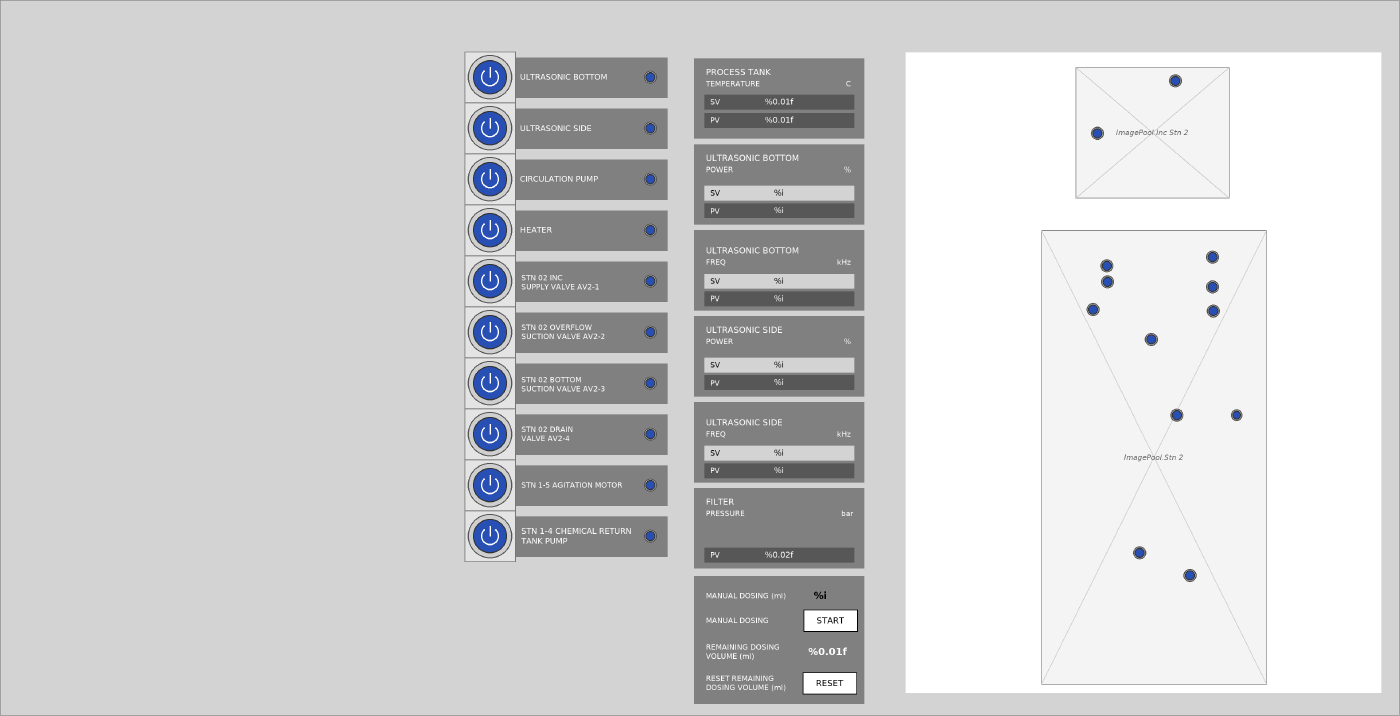
VISUALIZATION Manual_Station02  // 1920x983
    Rectangle (0,0 1920x983)
    Rectangle (1242,72 652x879)
    Image (1428,316 309x624), image: ImagePool.Stn 2
    RoundedRectangle (676,79 239x55)
    Label (710,98 163x16), "ULTRASONIC BOTTOM"
    Lamp1 (882,96 20x20), variable: ARdsMAP_HmiVariableStn[2].bProTankUsBtm_IND, style: Lamp-Lamp1-Blue
    PowerSwitch (637,71 70x70), variable: ARdsMAP_HmiVariableStn[2].bProTankUsBtm_PB, behaviour: TOGGLE, style: Switch-PowerSwitch-Blue
    RoundedRectangle (684,219 231x55)
    Label (710,228 161x36), "CIRCULATION PUMP"
    Lamp1 (882,236 20x20), variable: ARdsMAP_HmiVariableStn[2].bProTankPump_IND, style: Lamp-Lamp1-Blue
    PowerSwitch (637,211 70x70), variable: ARdsMAP_HmiVariableStn[2].bProTankPump_PB, behaviour: TOGGLE, style: Switch-PowerSwitch-Blue
    RoundedRectangle (684,289 231x55)
    Label (710,308 151x16), "HEATER"
    Lamp1 (882,306 20x20), variable: ARdsMAP_HmiVariableStn[2].bProTankHeater_IND, style: Lamp-Lamp1-Blue
    PowerSwitch (637,281 70x70), variable: ARdsMAP_HmiVariableStn[2].bProTankHeater_PB, behaviour: TOGGLE, style: Switch-PowerSwitch-Blue
    RoundedRectangle (684,429 231x55)
    Label (712,438 160x36), "STN 02 OVERFLOW SUCTION VALVE AV2-2"
    Lamp1 (882,446 20x20), variable: ARdsMAP_HmiVariableStn[2].bValve02_IND, style: Lamp-Lamp1-Blue
    PowerSwitch (637,421 70x70), variable: ARdsMAP_HmiVariableStn[2].bValve02_PB, behaviour: TOGGLE, style: Switch-PowerSwitch-Blue
    RoundedRectangle (684,359 231x55)
    Lamp1 (882,376 20x20), variable: ARdsMAP_HmiVariableStn[2].bValve01_IND, style: Lamp-Lamp1-Blue
    PowerSwitch (637,351 70x70), variable: ARdsMAP_HmiVariableStn[2].bValve01_PB, behaviour: TOGGLE, style: Switch-PowerSwitch-Blue
    Label (712,370 151x36), "STN 02 INC SUPPLY VALVE AV2-1"
    RoundedRectangle (676,149 239x55)
    Label (710,168 163x17), "ULTRASONIC SIDE"
    Lamp1 (882,166 20x20), variable: ARdsMAP_HmiVariableStn[2].bProTankUsSide_IND, style: Lamp-Lamp1-Blue
    PowerSwitch (637,141 70x70), variable: ARdsMAP_HmiVariableStn[2].bProTankUsSide_PB, behaviour: TOGGLE, style: Switch-PowerSwitch-Blue
    RoundedRectangle (684,569 231x55)
    Label (712,578 160x36), "STN 02 DRAIN VALVE AV2-4"
    Lamp1 (882,586 20x20), variable: ARdsMAP_HmiVariableStn[2].bValve04_IND, style: Lamp-Lamp1-Blue
    PowerSwitch (637,561 70x70), variable: ARdsMAP_HmiVariableStn[2].bValve04_PB, behaviour: TOGGLE, style: Switch-PowerSwitch-Blue
    RoundedRectangle (684,499 231x55)
    Lamp1 (882,516 20x20), variable: ARdsMAP_HmiVariableStn[2].bValve03_IND, style: Lamp-Lamp1-Blue
    PowerSwitch (637,491 70x70), variable: ARdsMAP_HmiVariableStn[2].bValve03_PB, behaviour: TOGGLE, style: Switch-PowerSwitch-Blue
    Label (712,510 151x36), "STN 02 BOTTOM SUCTION VALVE AV2-3"
    RoundedRectangle (684,639 231x55)
    Label (712,648 160x36), "STN 1-5 AGITATION MOTOR"
    Lamp1 (882,656 20x20), variable: ARdsMAP_HmiVariableGeneral.bProTankAgitationMotor_IND, style: Lamp-Lamp1-Blue
    PowerSwitch (637,631 70x70), variable: ARdsMAP_HmiVariableGeneral.bProTankAgitationMotor_PB, behaviour: TOGGLE, style: Switch-PowerSwitch-Blue
    RoundedRectangle (684,709 231x55)
    Label (712,718 160x36), "STN 1-4 CHEMICAL RETURN TANK PUMP"
    Lamp1 (882,726 20x20), style: Lamp-Lamp1-Blue
    PowerSwitch (637,701 70x70), variable: ARdsMAP_HmiVariableGeneral.bProTankPump_PB, behaviour: TOGGLE, style: Switch-PowerSwitch-Blue
    Lamp1 (1569,456 20x20), variable: ARdsMAP_HmiVariableStn[2].bProTankUsBtm_IND, style: Lamp-Lamp1-Blue
    Lamp1 (1553,749 20x20), variable: ARdsMAP_HmiVariableStn[2].bProTankPump_IND, style: Lamp-Lamp1-Blue
    Lamp1 (1509,377 20x20), variable: ARdsMAP_HmiVariableStn[2].bProTankHeater_IND, style: Lamp-Lamp1-Blue
    Lamp1 (1687,560 18x20), variable: ARdsMAP_HmiVariableStn[2].bValve02_IND, style: Lamp-Lamp1-Blue
    Lamp1 (1489,415 20x20), variable: ARdsMAP_HmiVariableStn[2].bProTankUsSide_IND, style: Lamp-Lamp1-Blue
    Lamp1 (1622,780 20x20), variable: ARdsMAP_HmiVariableStn[2].bValve04_IND, style: Lamp-Lamp1-Blue
    Lamp1 (1604,560 20x20), variable: ARdsMAP_HmiVariableStn[2].bValve03_IND, style: Lamp-Lamp1-Blue
    Lamp1 (1508,355 20x20), variable: ARdsMAP_HmiVariableStn[2].bProcessTankMinLevel_IND, style: Lamp-Lamp1-Blue
    Lamp1 (1653,343 20x20), variable: ARdsMAP_HmiVariableStn[2].bOverflowMaxLevel_IND, style: Lamp-Lamp1-Blue
    Lamp1 (1653,384 20x20), variable: ARdsMAP_HmiVariableStn[2].bOverflowMinLevel_IND, style: Lamp-Lamp1-Blue
    Lamp1 (1654,417 20x20), variable: ARdsMAP_HmiVariableStn[2].bProTankUsSide_IND, style: Lamp-Lamp1-Blue
    Image (1475,92 211x180), image: ImagePool.Inc Stn 2
    Lamp1 (1602,101 20x20), variable: ARdsMAP_HmiVariableStn[2].bValve01_IND, style: Lamp-Lamp1-Blue
    Lamp1 (1495,173 20x20), variable: ARdsMAP_HmiVariableStn[2].bDosingPump_IND, style: Lamp-Lamp1-Blue
    Group (952,791 233x175)
        RoundedRectangle (0,0 233x175)
        Rectangle (150,46 74x30), "START", colour toggle: ARbStnManualDosingST[2]
            toggle ARbStnManualDosingST[2]
        Label (13,47 109x28), "MANUAL DOSING"
        Label (13,13 121x28), "MANUAL DOSING (ml)"
        Rectangle (132,13 82x28), "%i", text variable: ARDSProminentDosingHMI[2].In_iManualDosingVolume_ml
            OnMouseDown: write the text variable via VisuDialogs.Numpad, min 1, max 32767
        Label (13,133 129x28), "RESET REMAINING DOSING VOLUME (ml)"
        Rectangle (149,132 74x30), "RESET", colour toggle: ARDSProminentDosingHMI[2].In_bResetRemainedDosingVolumePB
            tap ARDSProminentDosingHMI[2].In_bResetRemainedDosingVolumePB
        Label (13,90 118x28), "REMAINING DOSING VOLUME (ml)"
        Rectangle (142,90 82x28), "%0.01f", text variable: ARDSProminentDosingHMI[2].Out_rRemainedDosingVolume_ml
    RoundedRectangle (952,80 233x110)
    Label (1141,104 29x22), "C"
    Rectangle (966,130 205x20), "%0.01f", text variable: ARrStnTempSV[2]
    Label (971,129 22x22), "SV"
    Rectangle (966,155 205x20), "%0.01f", text variable: ARrStnTempPV[2]
    Label (971,154 22x22), "PV"
    Label (965,91 150x16), "PROCESS TANK"
    Label (965,104 99x22), "TEMPERATURE"
    RoundedRectangle (952,198 233x110)
    Label (1141,222 29x22), "%"
    Rectangle (966,255 205x20), "%i", text variable: ARiStnManualUSBtmAsv[2]
        OnMouseDown: write the text variable via VisuDialogs.Numpad, min 10, max 100
    Label (971,254 22x22), "SV"
    Rectangle (966,279 205x20), "%i", text variable: ARiStnUSBtmAPv[2]
    Label (971,279 22x22), "PV"
    Label (965,209 150x16), "ULTRASONIC BOTTOM"
    Label (965,222 99x22), "POWER"
    Group (952,670 233x110)
        RoundedRectangle (0,0 233x110)
        Label (189,24 32x22), "bar"
        Rectangle (14,82 205x20), "%0.02f", text variable: ARrStnFilterPressurePV[2]
        Label (19,81 22x22), "PV"
        Label (13,11 150x16), "FILTER"
        Label (13,24 99x22), "PRESSURE"
    Group (952,316 233x110)
        RoundedRectangle (0,0 233x110)
        Label (189,33 29x22), "kHz"
        Rectangle (14,84 205x20), "%i", text variable: ARiStnUSBtmAFreqPv[2]
        Label (19,83 22x22), "PV"
        Rectangle (14,60 205x20), "%i", text variable: DSWeberEnclosure[1].DSWeberGenerator[4].DSWeberMulFreqSwitching.iFreqOutput_TS
            tap DSWeberEnclosure[1].DSWeberGenerator[4].DSWeberMulFreqSwitching.bFreqSwitchingPB_TS
        Label (19,59 22x22), "SV"
        Label (13,33 99x22), "FREQ"
        Label (13,20 150x16), "ULTRASONIC BOTTOM"
    Group (952,434 233x110)
        RoundedRectangle (0,0 233x110)
        Label (189,24 29x22), "%"
        Rectangle (14,57 205x20), "%i", text variable: ARiStnManualUSSideAsv[2]
            OnMouseDown: write the text variable via VisuDialogs.Numpad, min 10, max 100
        Label (19,56 22x22), "SV"
        Rectangle (14,81 205x20), "%i", text variable: ARiStnUSSideAPv[2]
        Label (19,81 22x22), "PV"
        Label (13,11 150x16), "ULTRASONIC SIDE"
        Label (13,24 99x22), "POWER"
    Group (952,552 233x110)
        RoundedRectangle (0,0 233x110)
        Label (13,33 99x22), "FREQ"
        Label (13,20 150x16), "ULTRASONIC SIDE"
        Label (189,33 29x22), "kHz"
        Rectangle (14,84 205x20), "%i", text variable: ARiStnUSSideAFreqPv[2]
        Label (19,83 22x22), "PV"
        Rectangle (14,60 205x20), "%i", text variable: DSWeberEnclosure[1].DSWeberGenerator[3].DSWeberMulFreqSwitching.iFreqOutput_TS
            tap DSWeberEnclosure[1].DSWeberGenerator[3].DSWeberMulFreqSwitching.bFreqSwitchingPB_TS
        Label (19,59 22x22), "SV"
END_VISUALIZATION

(* stored: Version 1.1.0.1, ProductVersion 3.1.4024.12
   Visu Manual_Station02: Id {8d4c92f6-67c0-4ff2-afad-0ba40d2484cb} *)
